IF En THEN
	IF bError=FALSE THEN
		Channel_1_Output:=bDo_1;
		Channel_2_Output:=bDo_2;
		Channel_3_Output:=bDo_3;
		Channel_4_Output:=bDo_4;
		Channel_5_Output:=bDo_5;
		Channel_6_Output:=bDo_6;
		Channel_7_Output:=bDo_7;
		Channel_8_Output:=bDo_8;
		Channel_9_Output:=bDo_9;
		Channel_10_Output:=bDo_10;
		Channel_11_Output:=bDo_11;
		Channel_12_Output:=bDo_12;
		Channel_13_Output:=bDo_13;
		Channel_14_Output:=bDo_14;
		Channel_15_Output:=bDo_15;
		Channel_16_Output:=bDo_16;
	ELSE
		Channel_1_Output:=FALSE;
		Channel_2_Output:=FALSE;
		Channel_3_Output:=FALSE;
		Channel_4_Output:=FALSE;
		Channel_5_Output:=FALSE;
		Channel_6_Output:=FALSE;
		Channel_7_Output:=FALSE;
		Channel_8_Output:=FALSE;
		Channel_9_Output:=FALSE;
		Channel_10_Output:=FALSE;
		Channel_11_Output:=FALSE;
		Channel_12_Output:=FALSE;
		Channel_13_Output:=FALSE;
		Channel_14_Output:=FALSE;
		Channel_15_Output:=FALSE;
		Channel_16_Output:=FALSE;
	END_IF
END_IF

END_FUNCTION_BLOCK

// tc_mca_std_lib/POUs/Hardware/EtherCAT_Terminals/Measuring_Terminals/EL5002
//EL5002 | 2-chennel SSI absolute encoder terminal
FUNCTION_BLOCK EL5002

VAR_INPUT
	En: BOOL;
	iTerminal_ID : INT;
	ErrorSystem : POINTER TO ST_ErrorSystem;
END_VAR

VAR_OUTPUT
	EnO: BOOL;
	Ch1_Counter_Value : UDINT;
	Ch2_Counter_Value : UDINT;
	bError: BOOL;
END_VAR

VAR
	udi_Ch1_Cnt_Value AT %I* : UDINT;
	udi_Ch2_Cnt_Value AT %I* : UDINT;
	WcState_WcState AT %I*: BOOL;
	InfoData_State AT %I*: UINT;
	
	//FB-s
	EL5002_Error : FB_TerminalError;
END_VAR

(*
* TODO:
* Channel Status words
*)

EnO:=En;

//Error FB instance
EL5002_Error(
	En := TRUE,
	iTerminal_ID := iTerminal_ID,
	bWcState := WcState_WcState,
	uiInfoData_State := InfoData_State,
	pErrorSystem := ErrorSystem,
	bError => bError,
);

IF EN THEN
	IF NOT bError THEN
		Ch1_Counter_Value := udi_Ch1_Cnt_Value;
		Ch2_Counter_Value := udi_Ch2_Cnt_Value;
	ELSE
		Ch1_Counter_Value := 0;
		Ch2_Counter_Value := 0;
	END_IF
END_IF

END_FUNCTION_BLOCK

// tc_mca_std_lib/POUs/Hardware/EtherCAT_Terminals/Measuring_Terminals/EL5021
//EL5021 | 1-channel Sin/Cos encoder
FUNCTION_BLOCK EL5021

VAR_INPUT
	En: BOOL;
	iTerminal_ID : INT;
	ErrorSystem : POINTER TO ST_ErrorSystem;
END_VAR

VAR_OUTPUT
	EnO: BOOL;
	Counter_Value : UDINT;
	Latch_Value : UDINT;
	bError: BOOL;
END_VAR

VAR
	udiCounter_Value AT %I* : UDINT;
	udiLatch_Value AT %I* : UDINT;
	WcState_WcState AT %I*: BOOL;
	InfoData_State AT %I*: UINT;
	
	//FB-s
	EL5021_Error : FB_TerminalError;
END_VAR

(*
* TODO:
* Channel Status words, control words
*)

EnO:=En;

//Error FB instance
EL5021_Error(
	En := TRUE,
	iTerminal_ID := iTerminal_ID,
	bWcState := WcState_WcState,
	uiInfoData_State := InfoData_State,
	pErrorSystem := ErrorSystem,
	bError => bError,
);

IF EN THEN
	IF NOT bError THEN
		Counter_Value := udiCounter_Value;
		Latch_Value := udiLatch_Value;
	ELSE
		Counter_Value := 0;
		Latch_Value := 0;
	END_IF
END_IF

END_FUNCTION_BLOCK

// tc_mca_std_lib/POUs/Hardware/EtherCAT_Terminals/Measuring_Terminals/EL5042
//EL5042 | 2-channel BiSS-C absolute encoder terminal
FUNCTION_BLOCK EL5042

VAR_INPUT
	En: BOOL;
	iTerminal_ID : INT;
	ErrorSystem : POINTER TO ST_ErrorSystem;
END_VAR

VAR_OUTPUT
	EnO: BOOL;
	Ch1_Position : ULINT;
	Ch2_Position : ULINT;
	bError: BOOL;
END_VAR

VAR
	FB_Inputs_ch1_Position AT %I* : ULINT;
	FB_Inputs_ch2_Position AT %I* : ULINT;
	WcState_WcState AT %I*: BOOL;
	InfoData_State AT %I*: UINT;
	
	//FB-s
	EL5042_Error : FB_TerminalError;
END_VAR

(*
* TODO:
* Channel Status words
*)

EnO:=En;

//Error FB instance
EL5042_Error(
	En := TRUE,
	iTerminal_ID := iTerminal_ID,
	bWcState := WcState_WcState,
	uiInfoData_State := InfoData_State,
	pErrorSystem := ErrorSystem,
	bError => bError,
);

IF EN THEN
	IF NOT bError THEN
		Ch1_Position := FB_Inputs_ch1_Position;
		Ch2_Position := FB_Inputs_ch2_Position;
	ELSE
		Ch1_Position := 0;
		Ch2_Position := 0;
	END_IF
END_IF

END_FUNCTION_BLOCK

// tc_mca_std_lib/POUs/Hardware/EtherCAT_Terminals/Measuring_Terminals/EL5101
// EL5101 | 1-channel incremental encoder terminal, 5V, RS422
FUNCTION_BLOCK EL5101

VAR_INPUT
	En: BOOL;
	iTerminal_ID : INT;
	ErrorSystem : POINTER TO ST_ErrorSystem;
END_VAR

VAR_OUTPUT
	EnO: BOOL;
	Counter_Value : UINT;
	Latch_Value : UINT;
	bError: BOOL;
END_VAR

VAR
	uiCounter_Value AT %I* : UINT;
	uiLatch_Value AT %I* : UINT;
	WcState_WcState AT %I*: BOOL;
	InfoData_State AT %I*: UINT;
	
	//FB-s
	EL5101_Error : FB_TerminalError;
END_VAR

(*
* TODO:
* Channel Status word, control words
*)

EnO:=En;

//Error FB instance
EL5101_Error(
	En := TRUE,
	iTerminal_ID := iTerminal_ID,
	bWcState := WcState_WcState,
	uiInfoData_State := InfoData_State,
	pErrorSystem := ErrorSystem,
	bError => bError,
);

IF EN THEN
	IF NOT bError THEN
		Counter_Value := uiCounter_Value;
		Latch_Value := uiLatch_Value;
	ELSE
		Counter_Value := 0;
		Latch_Value := 0;
	END_IF
END_IF

END_FUNCTION_BLOCK

// tc_mca_std_lib/POUs/Hardware/EtherCAT_Terminals/Motion/EL7211_v1_00
///EL7211 | Servo motor termional 5 A
FUNCTION_BLOCK EL7211_v1_00
VAR_INPUT
	En: BOOL;
END_VAR
VAR_OUTPUT
	EnO: BOOL;

	bError: BOOL;
END_VAR
VAR
	WcState_WcState AT %I*: BOOL;
	InfoData_State AT %I*: UINT;
END_VAR

EnO:=En;

IF En AND (WcState_WcState OR InfoData_State<>16#8) THEN
	bError:=TRUE;
ELSE
	bError:=FALSE;
END_IF

END_FUNCTION_BLOCK

// tc_mca_std_lib/POUs/Hardware/EtherCAT_Terminals/Motion/EL9576_v1_00
///EL9576 | Brake terminal (vap and resistor)
FUNCTION_BLOCK EL9576_v1_00
VAR_INPUT
	En: BOOL;
END_VAR
VAR_OUTPUT
	EnO: BOOL;
	bError: BOOL;	
	OverTemperature: BOOL;
	I2TError : BOOL;
	I2TWarning : BOOL;
	OverVoltage  : BOOL;
	UnderVoltage : BOOL;
	ChopperOn : BOOL;
	DCLinkVoltage : LREAL;
	DutyCycle  : LREAL;
	ResistorCurrent : LREAL;
	
END_VAR
VAR
	BCTOverTemperature AT %I*: BOOL;
	BCTI2TError AT %I*: BOOL;
	BCTI2TWarning AT %I*: BOOL;
	BCTOverVoltage  AT %I*: BOOL;
	BCTUnderVoltage  AT %I*: BOOL;
	BCTChopperOn  AT %I*: BOOL;
	BCTDCLinkVoltage AT %I*: UDINT;
	BCTDutyCycle  AT %I*: USINT;
	BCTResistorCurrent AT %I*: UDINT;
	WcState_WcState AT %I*: BOOL;
	InfoData_State AT %I*: UINT;
	
END_VAR

EnO:=En;

IF En AND (WcState_WcState OR InfoData_State<>16#8 OR BCTI2TError OR BCTI2TWarning OR BCTOverTemperature OR BCTOverVoltage OR BCTUnderVoltage) THEN
	bError:=TRUE;
ELSE
	bError:=FALSE;
END_IF

OverTemperature:=BCTOverTemperature;
I2TError:=BCTI2TError;
I2TWarning:=BCTI2TWarning;
OverVoltage:=BCTOverVoltage;
UnderVoltage:=bctUnderVoltage;
ChopperOn:=bctChopperOn;
DCLinkVoltage:=UDINT_TO_LREAL(bctDCLinkVoltage);
DutyCycle:=USINT_TO_LREAL(BCTDutyCycle);
ResistorCurrent:=UDINT_TO_LREAL(BCTResistorCurrent);

END_FUNCTION_BLOCK

// tc_mca_std_lib/POUs/Hardware/EtherCAT_Terminals/System/EL9410
//EL9410 | E-Bus power supplier and refresher, diagnostics
FUNCTION_BLOCK EL9410

VAR_INPUT
	En: BOOL;
	iTerminal_ID : INT;
	ErrorSystem : POINTER TO ST_ErrorSystem;
END_VAR

VAR_OUTPUT
	EnO: BOOL;
	bError: BOOL;
END_VAR

VAR
	bStatus_Us_UV AT %I* : BOOL;
	bStatus_Up_UV AT %I* : BOOL;
	WcState_WcState AT %I*: BOOL;
	InfoData_State AT %I*: UINT;
	
	//FB-s
	EL9410_Error : FB_TerminalError;
END_VAR

(*
* TODO:
* Status bits
*)

EnO:=En;

//Error FB instance
EL9410_Error(
	En := TRUE,
	iTerminal_ID := iTerminal_ID,
	bWcState := WcState_WcState,
	uiInfoData_State := InfoData_State,
	pErrorSystem := ErrorSystem,
	bError => bError,
);

END_FUNCTION_BLOCK

// tc_mca_std_lib/POUs/Hardware/EtherCAT_Terminals/System/EL9505
//EL9505 | Power supply terminal 5V
FUNCTION_BLOCK EL9505

VAR_INPUT
	En: BOOL;
	iTerminal_ID : INT;
	ErrorSystem : POINTER TO ST_ErrorSystem;
END_VAR

VAR_OUTPUT
	EnO: BOOL;
	bError: BOOL;
END_VAR

VAR
	bStatus_Uo_Power_OK AT %I* : BOOL;
	bStatus_Uo_Overload AT %I* : BOOL;
	WcState_WcState AT %I*: BOOL;
	InfoData_State AT %I*: UINT;
	
	//FB-s
	EL9505_Error : FB_TerminalError;
END_VAR

(*
* TODO:
* Status bits
*)
EnO:=En;

//Error FB instance
EL9505_Error(
	En := TRUE,
	iTerminal_ID := iTerminal_ID,
	bWcState := WcState_WcState,
	uiInfoData_State := InfoData_State,
	pErrorSystem := ErrorSystem,
	bError => bError,
);

END_FUNCTION_BLOCK

// tc_mca_std_lib/POUs/Hardware/Other/EK1200
FUNCTION_BLOCK EK1200
VAR_INPUT
	En: BOOL;
END_VAR
VAR_OUTPUT
	EnO: BOOL;
END_VAR

EnO:=En;

END_FUNCTION_BLOCK

// tc_mca_std_lib/POUs/Motion/FB_NcAxis
///#########################################################
///Function block to communicate between Nc and Plc.
///
///	Library:		
///	Tc2_MC2.lib
///
///	Global Variables:
///	
///	Data types:
///	
///	External functions:
///
///###########################################################
FUNCTION_BLOCK FB_NcAxis
VAR
	sVersion: STRING:='1.0.0';
END_VAR
VAR_INPUT
	En: BOOL;
END_VAR
VAR_OUTPUT
	EnO: BOOL;
	bError: BOOL;
	Status: ST_AxisStatus;
END_VAR
VAR
	Axis: AXIS_REF;
	InfoData_State AT %I*: UINT;
END_VAR

EnO:=En;

IF En AND InfoData_State<>16#8 THEN
	bError:=TRUE;
ELSE
	bError:=FALSE;
END_IF

IF En THEN
	Axis.ReadStatus();
	Status:=Axis.Status;
END_IF

END_FUNCTION_BLOCK

// UnitTests/BasicTests
PROGRAM BasicTests
VAR
    Motor: DUT_MotionStage;
    fbMotion: FB_MotionStageSim;
    fbRequest: FB_MotionRequest;

    bError: BOOL;
    errState: MC_AxisStates;
END_VAR

fbRequest(stMotionStage := Motor);
fbMotion(stMotionStage := Motor);

CASE Motor.Axis.Status.MotionState OF
   MC_AXISSTATE_ERRORSTOP,
   MC_AXISSTATE_STOPPING,
   MC_AXISSTATE_HOMING,
   MC_AXISSTATE_DISCRETEMOTION,
   MC_AXISSTATE_CONTINOUSMOTION,
   MC_AXISSTATE_SYNCHRONIZEDMOTION:
        IF NOT Motor.bBrakeRelease THEN
            bError := TRUE;
            errState := Motor.Axis.Status.MotionState;
        END_IF
END_CASE

END_PROGRAM

// UnitTests/Interactive
PROGRAM Interactive
VAR
    bInit: BOOL := FALSE;

    M1: DUT_MotionStage;
    fbMotionStageSim: FB_MotionStageSim;
    nCounter: UINT;

    stOut: DUT_PositionState;
    fbGoOut: FB_PositionStateMove;
    bOut: BOOL;
    bGoOut: BOOL;
    stIn: DUT_PositionState;
    fbGoIn: FB_PositionStateMove;
    bIn: BOOL;
    bGoIn: BOOL;
    stUnsafe: DUT_PositionState;
    fbGoBad: FB_PositionStateMove;
    bHCF: BOOL;
    bGoHCF: BOOL;
END_VAR

BasicTests();

fbMotionStageSim(stMotionStage:=M1,
                 nEnableMode:=ENUM_StageEnableMode.DURING_MOTION);
nCounter := nCounter + 1;

IF NOT bInit THEN
    bInit := TRUE;

    stOut.sName := 'Out';
    stOut.fPosition := 100;
    stOut.fDelta := 20;
    stOut.fVelocity := 10;
    stOut.bValid := TRUE;
    stOut.bMoveOk := TRUE;

    stIn.sName := 'In';
    stIn.fPosition := 0;
    stIn.fDelta := 0.1;
    stIn.fVelocity := 5;
    stIn.bValid := TRUE;
    stIn.bMoveOk := TRUE;

    stUnsafe.sName := 'HCF';
    stUnsafe.fPosition := -999;
    stUnsafe.fDelta := 6;
    stUnsafe.fVelocity := 42;
    stUnsafe.bValid := TRUE;
    stUnsafe.bMoveOk := FALSE;
END_IF

fbGoOut(
    bExecute:=bGoOut,
    stMotionStage:=M1,
    stPositionState:=stOut,
    bAtState=>bOut);
fbGoIn(
    bExecute:=bGoIn,
    stMotionStage:=M1,
    stPositionState:=stIn,
    bAtState=>bIn);
fbGoBad(
    bExecute:=bGoHCF,
    stMotionStage:=M1,
    stPositionState:=stUnsafe,
    bAtState=>bHCF);

END_PROGRAM
